FUNCTION_BLOCK FB_SetSolenoid
VAR_INPUT
END_VAR
VAR_OUTPUT
END_VAR
VAR
END_VAR

METHOD AirDry : BOOL
VAR_INPUT
END_VAR
AirDry:= FALSE;

GVL_IO.gDigOutputs.bSolenoidValveA := FALSE;
GVL_IO.gDigOutputs.bSolenoidValveB := FALSE;
GVL_IO.gDigOutputs.bSolenoidValveC := TRUE;

GVL_Calibration.eLeakTestState := E_LeakTestState.IDLE;

AirDry := TRUE;
RETURN;
END_METHOD

METHOD HoldPressure : BOOL
VAR_INPUT
END_VAR
HoldPressure:= FALSE;

GVL_IO.gDigOutputs.bSolenoidValveA := TRUE;
GVL_IO.gDigOutputs.bSolenoidValveB := FALSE;
GVL_IO.gDigOutputs.bSolenoidValveC := FALSE;

GVL_Calibration.eLeakTestState := E_LeakTestState.HOLD_PRESSURE;

HoldPressure := TRUE;
RETURN;
END_METHOD

METHOD Idle : BOOL
VAR_INPUT
END_VAR
Idle:= FALSE;

GVL_IO.gDigOutputs.bSolenoidValveA := FALSE;
GVL_IO.gDigOutputs.bSolenoidValveB := FALSE;
GVL_IO.gDigOutputs.bSolenoidValveC := FALSE;

GVL_Calibration.eLeakTestState := E_LeakTestState.IDLE;

Idle := TRUE;
RETURN;
END_METHOD

METHOD PressureUp : BOOL
VAR_INPUT
END_VAR
PressureUp:= FALSE;

GVL_IO.gDigOutputs.bSolenoidValveA := TRUE;
GVL_IO.gDigOutputs.bSolenoidValveB := TRUE;
GVL_IO.gDigOutputs.bSolenoidValveC := FALSE;

GVL_Calibration.eLeakTestState := E_LeakTestState.PRESSURE_UP;

PressureUp := TRUE;
RETURN;
END_METHOD

END_FUNCTION_BLOCK

(* stored: Version 1.1.0.1, ProductVersion 3.1.4024.15
   POU FB_SetSolenoid: Id {2f71664d-ad34-48c2-8dc8-59f8d0fe2c84}, SpecialFunc None
   Method AirDry: Id {a8293fa8-9464-4f1f-ad94-3fb93520fc78}
   Method HoldPressure: Id {981066b5-d51f-42a3-860b-3eb971036e6b}
   Method Idle: Id {c8d592fb-4026-4675-95df-925b93b61cb8}
   Method PressureUp: Id {431bf55b-2b33-4299-9b61-7c5d049add12} *)
